PROGRAM Q9
VAR
	inputButton : BOOL := FALSE;
	inputReset	: BOOL := FALSE;
		
	timerStart	: BOOL := FALSE;
	timerRunning: BOOL := FALSE;
	Timer_On: TON;	
	timerCount	: TIME := T#0S;
	
	warning		: BOOL := FALSE;
	count_warn	: TIME := T#10S;
	output		: BOOL := FALSE;
	count_out	: TIME := T#15S;

END_VAR
VAR // added by the converter: edge detectors and wires of the graphical bodies
    _w1, _w2, _w3, _w4 : BOOL;
END_VAR

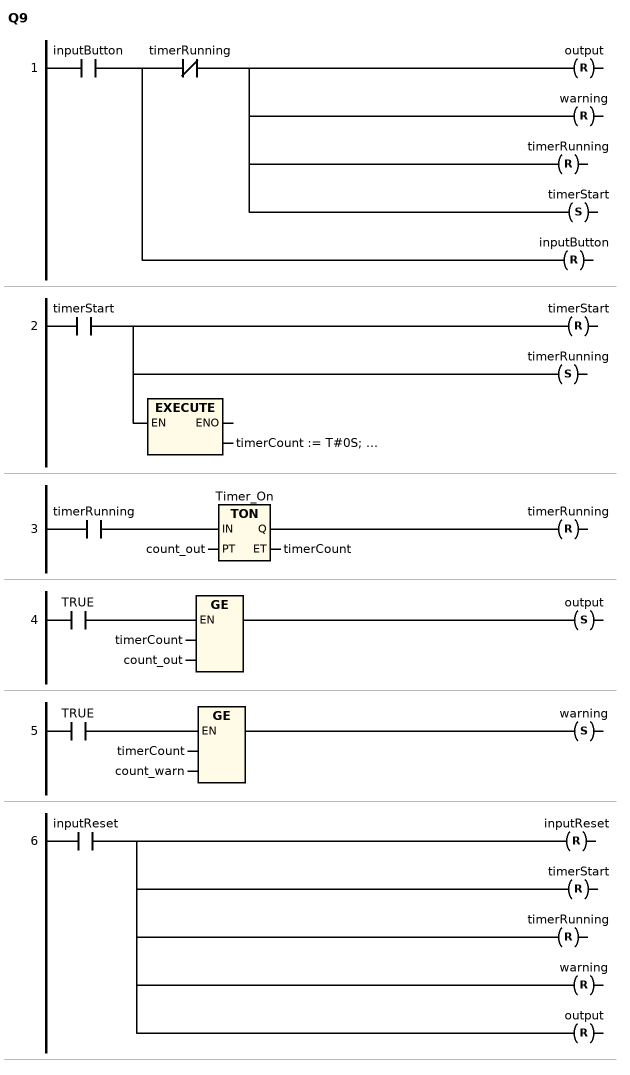
// NETWORK 1
_w1 := inputButton;
_w2 := _w1 AND NOT timerRunning;
output R= _w2;
warning R= _w2;
timerRunning R= _w2;
timerStart S= _w2;
inputButton R= _w1;

// NETWORK 2
_w3 := timerStart;
timerStart R= _w3;
timerRunning S= _w3;
IF _w3 THEN timerCount := T#0S; END_IF

// NETWORK 3
Timer_On(IN := timerRunning, PT := count_out, ET => timerCount); // TON
timerRunning R= Timer_On.Q;

// NETWORK 4
output S= timerCount >= count_out;

// NETWORK 5
warning S= timerCount >= count_warn;

// NETWORK 6
_w4 := inputReset;
inputReset R= _w4;
timerStart R= _w4;
timerRunning R= _w4;
warning R= _w4;
output R= _w4;

END_PROGRAM

(* stored: Version 1.1.0.1, ProductVersion 3.1.4024.12
   POU Q9: Id {fb09d2ad-996e-4d80-882a-44c8ce42b145}, SpecialFunc None *)
